FUNCTION_BLOCK BagView (* Composite Function Block Type *)
  (* Standard: 61499-2 *)
  (* Version 0.2, 2003-12-05, JHC, Rockwell Automation, Renamed from NEWCOMPFB. *)
  (* Version 0.1, 2002-01-08, JHC, Rockwell Automation, Added DLY FB as example. *)
  (* Version 0.0, 2000-05-27, JHC, Rockwell Automation *)
  (* Compiler header: package fb.rt.cs725;import fb.rt.vhmi.*; *)
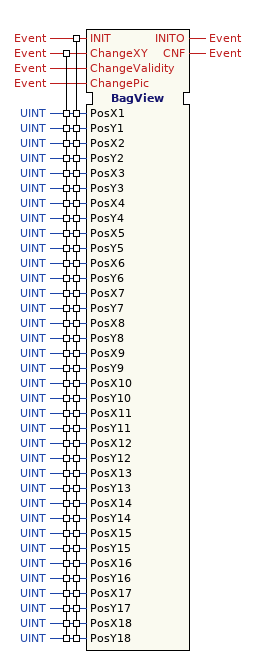
  EVENT_INPUT
    INIT WITH PosX1, PosY1, PosX2, PosY2, PosX3, PosY3, PosX4, PosY4, PosX5, PosY5, PosX6, PosY6, PosX7, PosY7, PosX8, PosY8, PosX9, PosY9, PosX10, PosY10, PosX11, PosY11, PosX12, PosY12, PosX13, PosY13, PosX14, PosY14, PosX15, PosY15, PosX16, PosY16, PosX17, PosY17, PosX18, PosY18; (* Initialization Request *)
    ChangeXY WITH PosX1, PosY1, PosX2, PosY2, PosX3, PosY3, PosX4, PosY4, PosX5, PosY5, PosX6, PosY6, PosX7, PosY7, PosX8, PosY8, PosX9, PosY9, PosX10, PosY10, PosX11, PosY11, PosX12, PosY12, PosX13, PosY13, PosX14, PosY14, PosX15, PosY15, PosX16, PosY16, PosX17, PosY17, PosX18, PosY18; (* Normal Execution Request *)
    ChangeValidity;
    ChangePic;
  END_EVENT
  EVENT_OUTPUT
    INITO; (* Initialization Confirm *)
    CNF; (* Execution Confirmation *)
  END_EVENT
  VAR_INPUT
    PosX1 : UINT;
    PosY1 : UINT;
    PosX2 : UINT;
    PosY2 : UINT;
    PosX3 : UINT;
    PosY3 : UINT;
    PosX4 : UINT;
    PosY4 : UINT;
    PosX5 : UINT;
    PosY5 : UINT;
    PosX6 : UINT;
    PosY6 : UINT;
    PosX7 : UINT;
    PosY7 : UINT;
    PosX8 : UINT;
    PosY8 : UINT;
    PosX9 : UINT;
    PosY9 : UINT;
    PosX10 : UINT;
    PosY10 : UINT;
    PosX11 : UINT;
    PosY11 : UINT;
    PosX12 : UINT;
    PosY12 : UINT;
    PosX13 : UINT;
    PosY13 : UINT;
    PosX14 : UINT;
    PosY14 : UINT;
    PosX15 : UINT;
    PosY15 : UINT;
    PosX16 : UINT;
    PosY16 : UINT;
    PosX17 : UINT;
    PosY17 : UINT;
    PosX18 : UINT;
    PosY18 : UINT;
  END_VAR
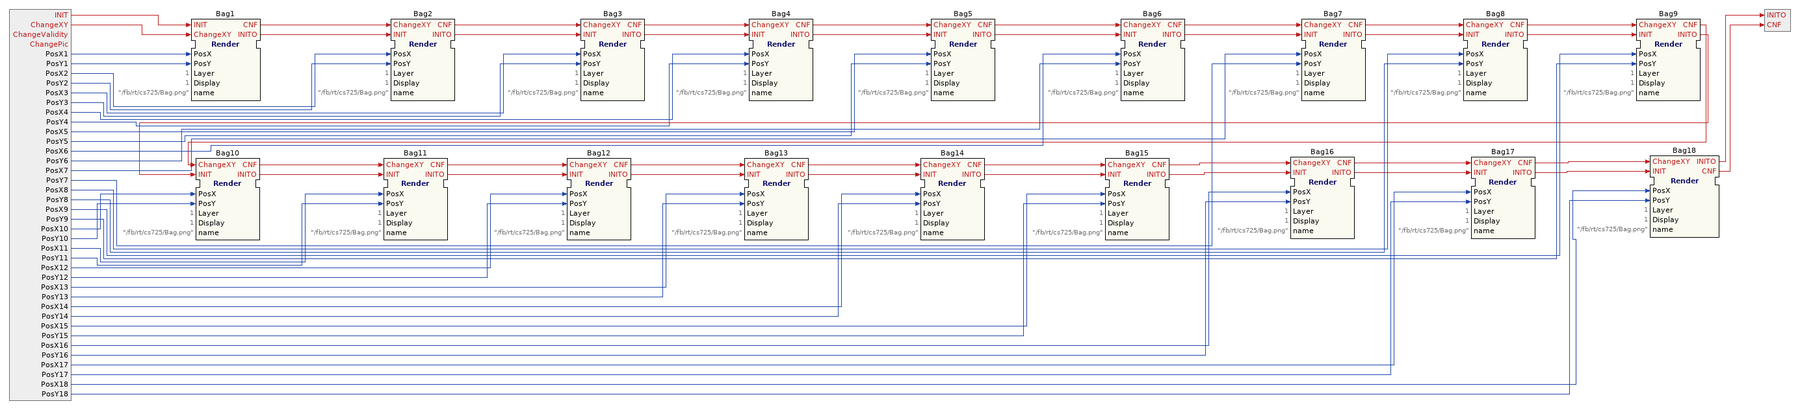
  FBS
    Bag1 : Render(Layer := 1, Display := 1, name := "/fb/rt/cs725/Bag.png");
    Bag2 : Render(Layer := 1, Display := 1, name := "/fb/rt/cs725/Bag.png");
    Bag3 : Render(Layer := 1, Display := 1, name := "/fb/rt/cs725/Bag.png");
    Bag4 : Render(Layer := 1, Display := 1, name := "/fb/rt/cs725/Bag.png");
    Bag5 : Render(Layer := 1, Display := 1, name := "/fb/rt/cs725/Bag.png");
    Bag6 : Render(Layer := 1, Display := 1, name := "/fb/rt/cs725/Bag.png");
    Bag7 : Render(Layer := 1, Display := 1, name := "/fb/rt/cs725/Bag.png");
    Bag8 : Render(Layer := 1, Display := 1, name := "/fb/rt/cs725/Bag.png");
    Bag9 : Render(Layer := 1, Display := 1, name := "/fb/rt/cs725/Bag.png");
    Bag10 : Render(Layer := 1, Display := 1, name := "/fb/rt/cs725/Bag.png");
    Bag11 : Render(Layer := 1, Display := 1, name := "/fb/rt/cs725/Bag.png");
    Bag12 : Render(Layer := 1, Display := 1, name := "/fb/rt/cs725/Bag.png");
    Bag13 : Render(Layer := 1, Display := 1, name := "/fb/rt/cs725/Bag.png");
    Bag14 : Render(Layer := 1, Display := 1, name := "/fb/rt/cs725/Bag.png");
    Bag15 : Render(Layer := 1, Display := 1, name := "/fb/rt/cs725/Bag.png");
    Bag16 : Render(Layer := 1, Display := 1, name := "/fb/rt/cs725/Bag.png");
    Bag17 : Render(Layer := 1, Display := 1, name := "/fb/rt/cs725/Bag.png");
    Bag18 : Render(Layer := 1, Display := 1, name := "/fb/rt/cs725/Bag.png");
  END_FBS
  EVENT_CONNECTIONS
    Bag1.CNF TO Bag2.ChangeXY;
    Bag2.CNF TO Bag3.ChangeXY;
    Bag3.CNF TO Bag4.ChangeXY;
    Bag4.CNF TO Bag5.ChangeXY;
    Bag5.CNF TO Bag6.ChangeXY;
    Bag6.CNF TO Bag7.ChangeXY;
    Bag7.CNF TO Bag8.ChangeXY;
    Bag8.CNF TO Bag9.ChangeXY;
    Bag9.CNF TO Bag10.ChangeXY;
    Bag10.CNF TO Bag11.ChangeXY;
    Bag11.CNF TO Bag12.ChangeXY;
    Bag12.CNF TO Bag13.ChangeXY;
    Bag13.CNF TO Bag14.ChangeXY;
    Bag14.CNF TO Bag15.ChangeXY;
    Bag15.CNF TO Bag16.ChangeXY;
    Bag16.CNF TO Bag17.ChangeXY;
    Bag17.CNF TO Bag18.ChangeXY;
    INIT TO Bag1.INIT;
    Bag1.INITO TO Bag2.INIT;
    Bag2.INITO TO Bag3.INIT;
    Bag3.INITO TO Bag4.INIT;
    Bag4.INITO TO Bag5.INIT;
    Bag5.INITO TO Bag6.INIT;
    Bag6.INITO TO Bag7.INIT;
    Bag7.INITO TO Bag8.INIT;
    Bag8.INITO TO Bag9.INIT;
    Bag9.INITO TO Bag10.INIT;
    Bag10.INITO TO Bag11.INIT;
    Bag11.INITO TO Bag12.INIT;
    Bag12.INITO TO Bag13.INIT;
    Bag13.INITO TO Bag14.INIT;
    Bag14.INITO TO Bag15.INIT;
    Bag15.INITO TO Bag16.INIT;
    Bag16.INITO TO Bag17.INIT;
    Bag17.INITO TO Bag18.INIT;
    Bag18.INITO TO INITO;
    Bag18.CNF TO CNF;
    ChangeXY TO Bag1.ChangeXY;
  END_CONNECTIONS
  DATA_CONNECTIONS
    PosX1 TO Bag1.PosX;
    PosY1 TO Bag1.PosY;
    PosX2 TO Bag2.PosX;
    PosY2 TO Bag2.PosY;
    PosX3 TO Bag3.PosX;
    PosY3 TO Bag3.PosY;
    PosX4 TO Bag4.PosX;
    PosY4 TO Bag4.PosY;
    PosX5 TO Bag5.PosX;
    PosY5 TO Bag5.PosY;
    PosX6 TO Bag6.PosX;
    PosY6 TO Bag6.PosY;
    PosX7 TO Bag7.PosX;
    PosY7 TO Bag7.PosY;
    PosX8 TO Bag8.PosX;
    PosY8 TO Bag8.PosY;
    PosX9 TO Bag9.PosX;
    PosY9 TO Bag9.PosY;
    PosX10 TO Bag10.PosX;
    PosY10 TO Bag10.PosY;
    PosX11 TO Bag11.PosX;
    PosY11 TO Bag11.PosY;
    PosX12 TO Bag12.PosX;
    PosY12 TO Bag12.PosY;
    PosX13 TO Bag13.PosX;
    PosY13 TO Bag13.PosY;
    PosX14 TO Bag14.PosX;
    PosY14 TO Bag14.PosY;
    PosX15 TO Bag15.PosX;
    PosY15 TO Bag15.PosY;
    PosX16 TO Bag16.PosX;
    PosY16 TO Bag16.PosY;
    PosX17 TO Bag17.PosX;
    PosY17 TO Bag17.PosY;
    PosX18 TO Bag18.PosX;
    PosY18 TO Bag18.PosY;
  END_CONNECTIONS
END_FUNCTION_BLOCK
